FUNCTION_BLOCK FbBlink (* Мигающий светодиод. *)
  (* Standard: 61499-1; Description: Мигающий светодиод. Simple FB with one algorithm *)
  (* Version 1.2, 2026-03-08, VA, LIB_PLC *)
  (* Documentation:
  // Мигающий светодиод. //            DbBlink //    +---------------------+ //    |       FbBlink       | //   -|TimeOn      BlinkLamp|->- //   -|TimeOff              | //   -|Ts_ms                | //   -|Reset                | //    +---------------------+ // Пример построения универсального кроссплатформенного графа состояний. // Использую этот код как заготовку под более сложные алгоритмы. // Данный алгоритм гораздо быстрее разрабатывать чем конечный автомат с памятью. // Граф состояний. // //            | //           -+- Reset //            | //            V //  +-------------------+ //  | State1 =          | //  | STATE_RESET       | //  | BlinkLamp = 0     | //  +-------------------+ //            | //            | //            | //            | //            V //  +-------------------+ //  | State1 =          | //  | STATE_ON          |<--------------+ //  | BlinkLamp = 1     |               | //  +-------------------+               | //            |                         | //            |                         | //           -+- Timer1 >= TimeOn      -+- Timer1 >= TimeOff //            |                         | //            V                         | //  +-------------------+               | //  | State1 =          |               | //  | STATE_OFF         |---------------+ //  | BlinkLamp = 0     | //  +-------------------+
  *)
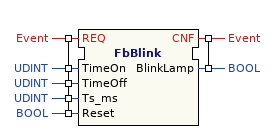
  EVENT_INPUT
    REQ WITH TimeOn, TimeOff, Ts_ms, Reset; (* Normal Execution Request *)
  END_EVENT
  EVENT_OUTPUT
    CNF WITH BlinkLamp; (* Execution Confirmation *)
  END_EVENT
  VAR_INPUT
    TimeOn : UDINT := 2000; (* Время включения лампочки [мс]. *)
    TimeOff : UDINT := 2000; (* Время выключения лампочки [мс]. *)
    Ts_ms : UDINT := 100; (* Шаг дискретизации по времени [мс]. *)
    Reset : BOOL := FALSE; (* Сброс при перезагрузке. *)
  END_VAR
  VAR_OUTPUT
    BlinkLamp : BOOL := FALSE; (* Мигающая лампочка. *)
  END_VAR
  VAR CONSTANT
    STATE_RESET : UINT := 0; (* Сброс при перезагрузке. *)
    STATE_ON : UINT := 1; (* Включить лампочку на заданное время. *)
    STATE_OFF : UINT := 2; (* Выключить лампочку на заданное время. *)
  END_VAR
  VAR
    Timer1 : UDINT := 0; (* Таймер1 [мс]. *)
    State1 : UINT := 0; (* Граф состояний. *)
  END_VAR
  EC_STATES
    REQ : REQ -> CNF;
  END_STATES
  ALGORITHM REQ IN ST:
IF (Reset) THEN // Сброс при перезагрузке.
	State1 := STATE_RESET;
END_IF;

CASE (State1) OF // Граф состояний.
	STATE_RESET : // Сброс.
		BlinkLamp := FALSE;
		Timer1 := 0;
		State1 := STATE_ON;

	STATE_ON : // Включить лампочку на заданное время.
		BlinkLamp := TRUE;
		Timer1 := Timer1 + Ts_ms;
		IF (Timer1 >= TimeOn) THEN
			State1 := STATE_OFF;
			Timer1 := 0;
		END_IF;

	STATE_OFF : // Выключить лампочку на заданное время.
		BlinkLamp := FALSE;
		Timer1 := Timer1 + Ts_ms;
		IF (Timer1 >= TimeOff) THEN
			State1 := STATE_ON;
			Timer1 := 0;
		END_IF;

	ELSE // RESET при неопределенном состоянии.
		State1 := STATE_RESET;
END_CASE; // CASE (State1) OF
  END_ALGORITHM
END_FUNCTION_BLOCK
